// TIA Portal project "2M-3" (V16)

(* hardware
DEVICE "S7-1200 station_1"  S7-1200 Station
   slot 0: "Rack_0"  S7-1200 Rack  Rack  V1.0
   slot 1: "PLC_1"  CPU 1212C AC/DC/Rly  6ES7 212-1BE40-0XB0  V4.0
*)

// ===== PLC "PLC_1"  CPU 1212C AC/DC/Rly =====

VAR_GLOBAL   // PLC tag table "Default tag table"
   "start" AT %I0.2 : Bool;
   "K1" AT %Q0.0 : Bool;
   "stop1" AT %I0.4 : Bool;
   "k2" AT %Q0.1 : Bool;
   "STOP" AT %I0.3 : Bool;
   "T1 tag" AT %M0.0 : Bool;
   "T2 tag" AT %M0.1 : Bool;
   "X" AT %M0.2 : Bool;
   "T3 tag" AT %M0.3 : Bool;
   "T4 tag" AT %M0.4 : Bool;
   "Tag_1" AT %M0.5 : Bool;
   "Tag_2" AT %M0.6 : Bool;
END_VAR

// folder: System blocks/Program resources

DATA_BLOCK "T1"   // DB2
{ S7_Optimized_Access := 'TRUE' }
AUTHOR : Simatic
FAMILY : IEC
NAME : IEC_TMR
VERSION : 1.0
// stored: InstanceOfName IEC_TIMER
"IEC_TIMER"
BEGIN
END_DATA_BLOCK

DATA_BLOCK "T2"   // DB3
{ S7_Optimized_Access := 'TRUE' }
AUTHOR : Simatic
FAMILY : IEC
NAME : IEC_TMR
VERSION : 1.0
// stored: InstanceOfName IEC_TIMER
"IEC_TIMER"
BEGIN
END_DATA_BLOCK

// folder: (top level)

ORGANIZATION_BLOCK "Main"   // OB1, LAD, ProgramCycle
TITLE = "Main Program Sweep (Cycle)"
{ S7_Optimized_Access := 'TRUE' }
VERSION : 0.1
   VAR_INPUT
      Initial_Call : Bool;   // Initial call of this OB
      Remanence : Bool;   // =True, if remanent data are available
   END_VAR
BEGIN

REGION Network 1: start
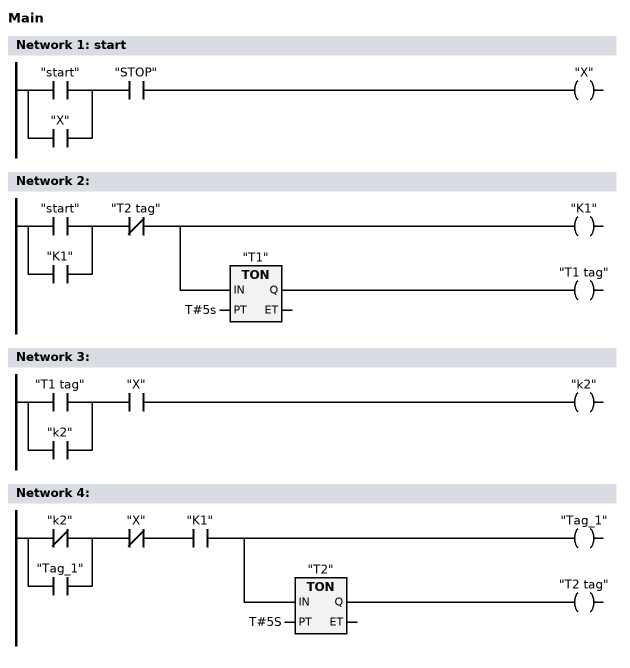
   RUNG wire#powerrail
      Contact( "start" )
      wire#w1
      Contact( "STOP" )
      Coil( "X" )
   END_RUNG
   RUNG wire#powerrail
      Contact( "X" )
   END_RUNG wire#w1
   // the same network as SCL:
   "X" := ("start" OR "X") AND "STOP";
END_REGION

REGION Network 2
   "K1" := ("start" OR "K1") AND NOT "T2 tag";
   "T1".TON(IN := "K1", PT := T#5s);
   "T1 tag" := "T1".Q;
END_REGION

REGION Network 3
   RUNG wire#powerrail
      Contact( "T1 tag" )
      wire#w1
      Contact( "X" )
      Coil( "k2" )
   END_RUNG
   RUNG wire#powerrail
      Contact( "k2" )
   END_RUNG wire#w1
   // the same network as SCL:
   "k2" := ("T1 tag" OR "k2") AND "X";
END_REGION

REGION Network 4
   "Tag_1" := (NOT "k2" OR "Tag_1") AND NOT "X" AND "K1";
   "T2".TON(IN := "Tag_1", PT := T#5S);
   "T2 tag" := "T2".Q;
END_REGION
END_ORGANIZATION_BLOCK